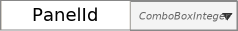
VISUALIZATION V_TpSelecCmb  // 238x31
    ComboBoxInteger (130,1 108x30), variable: VisuGVL.fbPanelImp.PanelId, text list: 'PanelCmbTxtList'
    Textfield (1,0 129x30), "PanelId"
END_VISUALIZATION

(* stored: Version 1.1.0.1, ProductVersion 3.1.4024.4
   Visu V_TpSelecCmb: Id {59a239aa-f142-4c88-83f5-fe1d59b1d714} *)
